{attribute 'strict'}
{attribute 'qualified_only'}
TYPE E_GantryMachineState :
(
	eIdle					:= 0,
	eAborting				:= 10,
	eAborted				:= 20,
	eStopping				:= 30,
	eStopped				:= 40,
	eStarting				:= 50,
	eRunning				:= 60,
	eReseting				:= 70,
	eRestarting				:= 80,
	eError					:= 1000	
);
END_TYPE

(* stored: Version 1.1.0.1, ProductVersion 3.1.4022.12
   DUT E_GantryMachineState: Id {e366e00e-7a9a-4580-a9e0-4f32496a74a4} *)
